FUNCTION TryConvert_LINT_TO_REAL : BOOL
VAR_INPUT
	in : LINT;
	out : REFERENCE TO REAL;
END_VAR

out := LINT_TO_REAL(in);
TryConvert_LINT_TO_REAL := TRUE;

END_FUNCTION

(* stored: Version 1.1.0.1, ProductVersion 3.1.4024.12
   POU TryConvert_LINT_TO_REAL: Id {668be3b1-4437-4e05-99de-695b01ce54ac}, SpecialFunc None *)
